// TwinCAT 3 PLC project TF8040_Template_Samples_PLC
// Title: TF8040 Template-Samples
// Company: Beckhoff Automation GmbH
// Author: Beckhoff Automation
// ProjectVersion: 2.0.0.0
// Description: Template-Samples to demonstrate the TF8040 PLC templates.
// ProgramVersion: 3.1.4023.0
// libraries:
//   Tc2_MDP, * (Beckhoff Automation GmbH)
//   Tc2_Standard, * (Beckhoff Automation GmbH)
//   Tc2_SUPS, * (Beckhoff Automation GmbH)
//   Tc2_System, * (Beckhoff Automation GmbH)
//   Tc2_Utilities, * (Beckhoff Automation GmbH)
//   Tc3_BA2, * (Beckhoff Automation GmbH)
//   Tc3_BA2_Common, * (Beckhoff Automation GmbH)
//   Tc3_BACnetRev14, * (Beckhoff Automation GmbH)
//   Tc3_Module, * (Beckhoff Automation GmbH)
//   Tc3_XBA, * (Beckhoff Automation GmbH)
// project tree:
//   / PlcTask.TcTTO (not stored)
//   POUs/ MAIN.TcPOU
//   Templates/DUTs/Enumerations/Building/ E_BA_BuildingMode.TcDUT
//   Templates/DUTs/Enumerations/Plant/AC/ E_BA_AC_OpMod01.TcDUT, E_BA_AC_SelSpErc.TcDUT
//   Templates/DUTs/Enumerations/Universal/ E_BA_EnergyLvl.TcDUT, E_BA_EnergyLvlA.TcDUT, E_BA_MdltCmd.TcDUT, E_BA_OnOff.TcDUT, E_BA_OnOffA.TcDUT
//   Templates/DUTs/Types/Building/ ST_BA_BuildingAlarms.TcDUT
//   Templates/DUTs/Types/General/ ST_BA_GeneralSettings.TcDUT
//   Templates/DUTs/Types/WeatherStation/ ST_BA_WeatherStation.TcDUT
//   Templates/GVLs/ BA2_Param.TcGVL
//   Templates/GVLs/DPAD/Labels/Composition/ LblCmpAC.TcGVL, LblCmpGeneral.TcGVL, LblCmpHeating.TcGVL, LblCmpRoomAutomation.TcGVL, LblUniControl.TcGVL, LblUniFieldDevice.TcGVL
//   Templates/GVLs/EventClasses/ EC_ID.TcGVL
//   Templates/GVLs/Language/English/ LblAggregates_EN.TcGVL, LblControl_EN.TcGVL, LblFunctions_EN.TcGVL, TxtEvent_EN.TcGVL, TxtPlant_EN.TcGVL, TxtTrade_EN.TcGVL
//   Templates/GVLs/Language/German/ LblAggregates_DE.TcGVL, LblControl_DE.TcGVL, LblFunctions_DE.TcGVL, TxtEvent_DE.TcGVL, TxtPlant_DE.TcGVL, TxtTrade_DE.TcGVL
//   Templates/GVLs/Site/ Site.TcGVL
//   Templates/POUs/Trade/AC/Aggregates/Cooler/Temperature/ FB_BA_AC_ColTSuACtrl.TcPOU, FB_BA_AC_ColT_02.TcPOU
//   Templates/POUs/Trade/AC/Aggregates/ERC/ FB_BA_AC_ErcTSuACtrl.TcPOU
//   Templates/POUs/Trade/AC/Aggregates/ERC/Plate/ FB_BA_AC_ErcPl_02.TcPOU
//   Templates/POUs/Trade/AC/Aggregates/PreHeater/ FB_BA_AC_PreHtr.TcPOU, FB_BA_AC_PreHtrTSuACtrl.TcPOU, FB_BA_AC_TRtCtrl.TcPOU
//   Templates/POUs/Trade/AC/ FB_BA_AC.TcPOU
//   Templates/POUs/Trade/AC/General/ FB_BA_AC_OpMod1St.TcPOU, FB_BA_AC_SumNgtCol.TcPOU
//   Templates/POUs/Trade/AC/Plants/ FB_BA_AHU_1st_10.TcPOU
//   Templates/POUs/Trade/AC/Setpoint/Temperature/ FB_BA_AC_SpTRm_01.TcPOU, FB_BA_AC_TCasCtrl_01.TcPOU
//   Templates/POUs/Trade/General/Building/ FB_BA_BuildingAlarms.TcPOU, FB_BA_BuildingGlobal.TcPOU, FB_BA_BuildingMode.TcPOU
//   Templates/POUs/Trade/General/ControlCabinet/ FB_BA_ControlCabinet.TcPOU, FB_BA_ControlCabinetBasic.TcPOU
//   Templates/POUs/Trade/General/EventClasses/ FB_BA_EvtGroups.TcPOU
//   Templates/POUs/Trade/General/ FB_BA_General.TcPOU
//   Templates/POUs/Trade/General/IFP/ FB_BA_IFP.TcPOU
//   Templates/POUs/Trade/General/IFP/Project/ FB_BA_ProjectEx.TcPOU
//   Templates/POUs/Trade/General/Settings/ FB_BA_Settings.TcPOU, FB_BA_WeatherParamter.TcPOU
//   Templates/POUs/Trade/HeatingSystem/Distribution/HeatingCircuit/ FB_BA_H_HtgCir01.TcPOU
//   Templates/POUs/Trade/HeatingSystem/ FB_BA_H.TcPOU
//   Templates/POUs/Trade/HeatingSystem/General/ FB_BA_HtgLmt.TcPOU, FB_BA_H_OpMod.TcPOU
//   Templates/POUs/Trade/HeatingSystem/Setpoint/ FB_BA_H_HtgCir_Sp.TcPOU
//   Templates/POUs/Trade/OutdoorDevices/ FB_BA_OD.TcPOU
//   Templates/POUs/Trade/OutdoorDevices/WeatherStation/ FB_BA_WeatherStation_Draft.TcPOU
//   Templates/POUs/Universal/Aggregat/Analog/ FB_BA_ActuatorAnalog.TcPOU
//   Templates/POUs/Universal/Aggregat/Binary/ FB_BA_ActuatorCmd.TcPOU
//   Templates/POUs/Universal/Control/AntiBlocking/ FB_BA_AntiBlocking.TcPOU
//   Templates/POUs/Universal/Control/EventClasses/ FB_BA_EvtCategory.TcPOU
//   Templates/POUs/Universal/Control/Hysteresis/ FB_BA_Hys_21.TcPOU
//   Templates/POUs/Universal/Control/Monitoring/ FB_BA_FdbAnalog.TcPOU, FB_BA_FdbBinary.TcPOU
//   Templates/POUs/Universal/Control/PID/ FB_BA_PID.TcPOU, FB_BA_PID_Sp.TcPOU
//   Templates/POUs/Universal/Control/Ramp/ FB_BA_RampLimitIncrease.TcPOU
//   Templates/POUs/Universal/Control/Scale/ FB_BA_Scale_02.TcPOU, FB_BA_Scale_04.TcPOU, FB_BA_Scale_04_Y2_3.TcPOU (not stored)
//   Templates/POUs/Universal/Control/TimeDelay/ FB_BA_DlyOff.TcPOU, FB_BA_DlyOn.TcPOU
//   Templates/POUs/Universal/Control/Trend/ FB_BA_TrendLogging.TcPOU
//   Templates/POUs/Universal/Damper/2P/ FB_BA_Dmp2P.TcPOU
//   Templates/POUs/Universal/Motor/1st/ FB_BA_Mot1st.TcPOU
//   Templates/POUs/Universal/Motor/Control/ FB_BA_MotCtlExt.TcPOU
//   Templates/POUs/Universal/Pump/1st/ FB_BA_Pu1st.TcPOU
//   Templates/POUs/Universal/Sensor/ FB_BA_CombinationBI_BV.TcPOU, FB_BA_MeasuredValueCardinal.TcPOU, FB_BA_SensorAnalog.TcPOU, FB_BA_SensorAnalog_IO.TcPOU, FB_BA_SensorBinary.TcPOU, FB_BA_SensorBinary_IO.TcPOU
//   Templates/POUs/Universal/Valve/ FB_BA_Vlv.TcPOU

// ---- Templates/DUTs/Enumerations/Building/E_BA_BuildingMode.TcDUT
{region '#Template'}
	{attribute 'Version' := '1.2.0.0'}
	{attribute 'Tags' := '"LCID": "1031", "Text": "DUT, Building, RA, OpMod, Mode"'}
	{attribute 'Tags' := '"LCID": "1033", "Text": "DUT, Building, RA, OpMod, Mode"'}
	{attribute 'Description' := '"LCID": "1031", "Text": "Gebäude-Betriebsart"'}
	{attribute 'Description' := '"LCID": "1033", "Text": "Building-operation-mode"'}
{endregion}

{attribute qualified_only}
TYPE E_BA_BuildingMode :
(
	eDefault		:= 1,
	eNightWatch		:= 2,
	eCleaning		:= 3
	
) UDINT;
END_TYPE

// ---- Templates/DUTs/Enumerations/Plant/AC/E_BA_AC_OpMod01.TcDUT
{region '#Template'}
	{attribute 'Version' := '1.0.0.0'}
	{attribute 'Tags' := '"LCID": "1031", "Text": "DUT, Plant, AC, OpMod"'}
	{attribute 'Tags' := '"LCID": "1033", "Text": "DUT, Plant, AC, OpMod"'}
	{attribute 'Description' := '"LCID": "1031", "Text": "Betriebsart Klimaanlage"'}
	{attribute 'Description' := '"LCID": "1033", "Text": "Operation Mode Air Conditioning"'}
{endregion}

{attribute qualified_only}
TYPE E_BA_AC_OpMod01 :
(
    Invalid							:= 0,
    eOff							:= 1,	// Aus							// Off
	eOn								:= 2,	// Ein							// On
    eEmergency						:= 3,	// Notfall						// Emergency
    eFrost							:= 4,	// Frost						// Frost
    eSmokeExtractionProgramm		:= 5,	// Entrauchung Programm			// Smoke extraction programm
    eSmokeExtractionSupplyAir		:= 6,	// Entrauchung Zuluft			// Smoke extraction supply air
    eSmokeExtractionExhaustAir		:= 7,	// Entrauchung Fortluft			// Smoke extraction exhaust air
    eFire							:= 8,	// Feuer						// Fire
    eNightCooling					:= 9,	// Nachtkühlung					// Night cooling
    eCoolDownProtection				:= 10,	// Stützbetrieb,Auskühlschutz	// Cool down protection
    eOverHeatingProtection			:= 11,	// Überhitzungsschutz			// Over heating protection
    eAlarm							:= 12,	// Störung						// Alarm
    eForcedVentilation				:= 13,	// Zwangsbelüftung				// Forced ventilation
    eCentralSwitchOff				:= 14	// Zentralabschaltung			// Central switch-off
) UDINT;
END_TYPE

// ---- Templates/DUTs/Enumerations/Plant/AC/E_BA_AC_SelSpErc.TcDUT
{region '#Template'}
	{attribute 'Version' := '1.0.0.0'}
	{attribute 'Tags' := '"LCID": "1031", "Text": "DUT, Plant, AC, Setpoint"'}
	{attribute 'Tags' := '"LCID": "1033", "Text": "DUT, Plant, AC, Setpoint"'}
	{attribute 'Description' := '"LCID": "1031", "Text": "Auswahl Sollwert Energie Rückgewinnung"'}
	{attribute 'Description' := '"LCID": "1033", "Text": "Selection setpoint energy recovery"'}
{endregion}

{attribute 'qualified_only'}
TYPE E_BA_AC_SelSpErc :
(
	eAction				:= 1,	//	E_BA_Action.eDirect = SpCol, E_BA_Action.eReverse = SpHtg, 
	eAverageHtgCol		:= 2	
) UDINT;
END_TYPE

// ---- Templates/DUTs/Enumerations/Universal/E_BA_EnergyLvl.TcDUT
{region '#Template'}
	{attribute 'Version' := '1.0.0.0'}
	{attribute 'Tags' := '"LCID": "1031", "Text": "DUT, Room automation, Heating system"'}
	{attribute 'Tags' := '"LCID": "1033", "Text": "DUT, Room automation, Heating system"'}
	{attribute 'Description' := '"LCID": "1031", "Text": "Betriebsart Energieniveau"'}
	{attribute 'Description' := '"LCID": "1033", "Text": "Operating mode Energy level"'}
{endregion}

{attribute qualified_only}
TYPE E_BA_EnergyLvl :
(
	eProtection		:= 1,
	eEconomy		:= 2,
	eComfort		:= 3
	
) UDINT;
END_TYPE

// ---- Templates/DUTs/Enumerations/Universal/E_BA_EnergyLvlA.TcDUT
{region '#Template'}
	{attribute 'Version' := '1.0.0.0'}
	{attribute 'Tags' := '"LCID": "1031", "Text": "DUT, Room automation, Heating system"'}
	{attribute 'Tags' := '"LCID": "1033", "Text": "DUT, Room automation, Heating system"'}
	{attribute 'Description' := '"LCID": "1031", "Text": "Betriebsart Energieniveau"'}
	{attribute 'Description' := '"LCID": "1033", "Text": "Operating mode Energy level"'}
{endregion}

{attribute qualified_only}
TYPE E_BA_EnergyLvlA :
(
	eAutomatic		:= 1,
	eProtection		:= 2,
	eEconomy		:= 3,
	eComfort		:= 4
	
) UDINT;
END_TYPE

// ---- Templates/DUTs/Enumerations/Universal/E_BA_MdltCmd.TcDUT
{region '#Template'}
	{attribute 'Version' := '1.0.0.0'}
	{attribute 'Tags' := '"LCID": "1031", "Text": "DUT, Operation mode, Universal, Modulation"'}
	{attribute 'Tags' := '"LCID": "1033", "Text": "DUT, Operation mode, Universal, Modulation"'}
	{attribute 'Description' := '"LCID": "1031", "Text": "Modulationsbefehle"'}
	{attribute 'Description' := '"LCID": "1033", "Text": "modulation commands"'}
{endregion}

{attribute 'qualified_only'}
TYPE E_BA_MdltCmd :
(
	eOff			:= 1,
	eOn				:= 2,
	eMin			:= 3,
	eMax			:= 4
	
) UDINT;
END_TYPE

// ---- Templates/DUTs/Enumerations/Universal/E_BA_OnOff.TcDUT
{region '#Template'}
	{attribute 'Version' := '1.0.0.0'}
	{attribute 'Tags' := '"LCID": "1031", "Text": "DUT, Operation mode, Universal, On, Off"'}
	{attribute 'Tags' := '"LCID": "1033", "Text": "DUT, Operation mode, Universal, On, Off"'}
	{attribute 'Description' := '"LCID": "1031", "Text": "Betriebsart Ein Aus"'}
	{attribute 'Description' := '"LCID": "1033", "Text": "Operating on off"'}
{endregion}

{attribute qualified_only}
TYPE E_BA_OnOff :
(
	eOff			:= 1,
	eOn				:= 2
	
) UDINT;
END_TYPE

// ---- Templates/DUTs/Enumerations/Universal/E_BA_OnOffA.TcDUT
{region '#Template'}
	{attribute 'Version' := '1.0.0.0'}
	{attribute 'Tags' := '"LCID": "1031", "Text": "DUT, Operation mode, Universal, On, Off"'}
	{attribute 'Tags' := '"LCID": "1033", "Text": "DUT, Operation mode, Universal, On, Off"'}
	{attribute 'Description' := '"LCID": "1031", "Text": "Betriebsart Ein Aus Auto"'}
	{attribute 'Description' := '"LCID": "1033", "Text": "Operating on off auto"'}
{endregion}

{attribute qualified_only}
TYPE E_BA_OnOffA :
(
	eAutomatic		:= 1,
	eOff			:= 2,
	eOn				:= 3
	
) UDINT;
END_TYPE

// ---- Templates/DUTs/Types/Building/ST_BA_BuildingAlarms.TcDUT
{region '#Template'}
	{attribute 'Version' := '1.2.0.0'}
	{attribute 'Tags' := '"LCID": "1031", "Text": "Types, Publisher, Subscriber, Building, General, Alarms, Events"'}
	{attribute 'Tags' := '"LCID": "1033", "Text": "Types, Publisher, Subscriber, Building, General, Alarms, Events"'}
	{attribute 'Description' := '"LCID": "1031", "Text": "Gebäude-Alarme und -Events"'}
	{attribute 'Description' := '"LCID": "1033", "Text": "Building-alarms and -events"'}
{endregion}
TYPE ST_BA_BuildingAlarms :
STRUCT
	bBurglary				: BOOL;
	bFireAlert				: BOOL;
	bCentralOff				: BOOL;
	bForcedVentilation		: BOOL;
	bSmokeExtraction		: BOOL;
END_STRUCT
END_TYPE

// ---- Templates/DUTs/Types/General/ST_BA_GeneralSettings.TcDUT
{region '#Template'}
	{attribute 'Version' := '1.0.0.0'}
	{attribute 'Tags' := '"LCID": "1031", "Text": "Types, Publisher, Subscriber, AC, General, Settings"'}
	{attribute 'Tags' := '"LCID": "1033", "Text": "Types, Publisher, Subscriber, AC, General, Settings"'}
	{attribute 'Description' := '"LCID": "1031", "Text": "Basis Daten AC"'}
	{attribute 'Description' := '"LCID": "1033", "Text": "Basic data AC"'}
{endregion}
TYPE ST_BA_GeneralSettings :
STRUCT
	fFrostProtectionSetpoint			: REAL;  // frost protection setpoint. for eg. Heating circutis in protection mode
	fTWth								: REAL;  // present value of outside temperature

	fTWthLowLimit						: REAL;  // below this value all frostprotection funcktions in HVAC-Plants will be enabled
	bTWthLowLimit						: BOOL;  // is TRUE when the outside temperature is below the value from fTWthLmtCrit 

	fTWthDamped							: REAL;  // damped outside temperature
	bTWthDampedLowLimit					: BOOL;  // is TRUE when the damped outside temperature is below the value from fTWthLmtCrit 

END_STRUCT
END_TYPE

// ---- Templates/DUTs/Types/WeatherStation/ST_BA_WeatherStation.TcDUT
{region '#Template'}
	{attribute 'Version' := '1.2.0.0'}
	{attribute 'Tags' := '"LCID": "1031", "Text": "Types, Publisher, Subscriber, Weather, Data"'}
	{attribute 'Tags' := '"LCID": "1033", "Text": "Types, Publisher, Subscriber, Weather, Data"'}
	{attribute 'Description' := '"LCID": "1031", "Text": "Daten Wetterstation"'}
	{attribute 'Description' := '"LCID": "1033", "Text": "Weatherstation-data"'}
{endregion}
TYPE ST_BA_WeatherStation :
STRUCT
	bDisturb				: BOOL;
	fLatitude				: REAL;				// [°]
	fLongitude				: REAL;				// [°]
	fSunAzimuth				: REAL;				// [°]
	fSunElevation			: REAL;				// [°]
	bRain					: BOOL;
	stDateTime				: TIMESTRUCT;
	fOutsideTemperature		: REAL;				// [°C]
	fDewPointTemperature	: REAL;				// [°C]		 
	fPressureAbs			: REAL;				// [hPa]
	fPressureRel			: REAL;				// [hPa]			 
	fHumidityAbs			: REAL;				// [g/m³]
	fHumidityRel			: REAL;				// [%rF]	
	fBrightnessNorth		: REAL;				// [Lux]		 
	fBrightnessEast			: REAL;				// [Lux]
	fBrightnessSouth		: REAL;				// [Lux]
	fBrightnessWest			: REAL;				// [Lux]			 
	fDawn					: REAL;				// [Lux] 
	fGlobalRadiation		: REAL;				// [W/m²]			 
	fWindDirection			: REAL;				// [°]
	fWindSpeed				: REAL;				// [m/s]
END_STRUCT
END_TYPE

// ---- Templates/GVLs/BA2_Param.TcGVL
{region '#Template'}
	{attribute 'Version' := '0.0.1.0'}
	{attribute 'Tags' := '"LCID": "1031", "Text": "GVL, Constants"'}
	{attribute 'Tags' := '"LCID": "1033", "Text": "GVL, Constants"'}
	{attribute 'Description' := '"LCID": "1031", "Text": "Globale Konstanten"'}
	{attribute 'Description' := '"LCID": "1033", "Text": "Global constants"'}
{endregion}

{attribute 'qualified_only'}
{attribute 'strict'}
VAR_GLOBAL CONSTANT 
	fAP                					: REAL 						:= 1013.25;	// Hydrostatischer Luftdruck	//	atmospheric pressure

	nDefTimeDelay_ToAbnormal			: UDINT						:= 1;
	nDefTimeDelay_ToNormal				: UDINT						:= 0;

	fDefCOVIncrement					: REAL						:= 0.1;	

	fDefLimitDeadband					: REAL						:= 0.0;

	nLoop_DefOpMode						: E_BA_PIDMode				:= E_BA_PIDMode.eP1ID;	
	
	{warning disable C0228}
	stTrend_DefStartTime				: ST_BA_DateTime			;(*:= F_BA_ToSTDateTime(DT#2099-01-01-00:13);*)
	stTrend_DefStopTime					: ST_BA_DateTime			;(* := F_BA_ToSTDateTime(DT#2099-01-01-00:13);*)
	{warning restore C0228}
	nTrend_BufferSize					: UDINT						:= 500;	// Count of entries in a Trend-Buffer	
	bTrend_DefLogEnable					: BOOL						:= FALSE;
	bTrend_DefStopOnFull				: BOOL						:= FALSE;
	nTrend_DefLogInterval				: UDINT						:= 90;	// (in [s])
	nTrend_DefNotificationThreshold		: UDINT						:= 50;
	eTrend_DefLoggingType				: E_BA_LoggingType			:= E_BA_LoggingType.ePolled;				
END_VAR

// ---- Templates/GVLs/DPAD/Labels/Composition/LblCmpAC.TcGVL
{region '#Template'}
	{attribute 'Version' := '1.2.0.0'}
	{attribute 'Tags' := '"LCID": "1031", "Text": "GVL, AC, AKS, Plants, ObjectName, Description"'}
	{attribute 'Tags' := '"LCID": "1033", "Text": "GVL, AC, DPAD, Plants, ObjectName, Description"'}
	{attribute 'Description' := '"LCID": "1031", "Text": "Anlagenkennzeichnungssystem, AC Labels Kompensation"'}
	{attribute 'Description' := '"LCID": "1033", "Text": "Data Point Addressing Description, AC labels compensation"'}
{endregion}

{attribute 'qualified_only'}
VAR_GLOBAL
///////////////////////
//	Aggregates\Cooler	
	Cooler_TFl							:FB_BA_Label	:= LblAggregates_TemperatureFlow;	
	Cooler_TRt							:FB_BA_Label	:= LblAggregates_TemperatureReturnFlow;	

	Cooler_TSuACtrl						:FB_BA_Label	:= LblControl_SupplyAirTemperatureControl;
	Cooler_TSuACtrl_Ctrl				:FB_BA_Label	:= LblFunctions_LoopObject; 
	Cooler_TSuALimitationCtrl			:FB_BA_Label	:= LblControl_SupplyAirTemperatureLimitationControl;

	Cooler_XSuACtrl						:FB_BA_Label	:= LblControl_SupplyAirDehumidifierControl; 
	Cooler_XSuACtrl_Ctrl				:FB_BA_Label	:= LblFunctions_LoopObject; 
	Cooler_Dehumf						:FB_BA_Label	:= LblControl_OperationalMessageDehumidification;	

	Cooler_Vlv							:FB_BA_Label	:= LblAggregates_Valve;
	Cooler_Pu							:FB_BA_Label	:= LblAggregates_Pump;
	
//	Aggregates\ERC
	ERC_DiffPrssSwi						:FB_BA_Label	:= LblAggregates_PressureDifferential;												 										 
	ERC_IcePrtcRamp						:FB_BA_Label	:= LblControl_EnergyRecoveryDeicingRamp;
	ERC_Motor							:FB_BA_Label	:= LblAggregates_HeatRecovery;
	ERC_TExhACtrl						:FB_BA_Label	:= LblControl_ExhaustAirTemperatureControl;
	ERC_TSuACtrl						:FB_BA_Label	:= LblControl_SupplyAirTemperatureControl;
	ERC_TSuACtrl_Ctrl					:FB_BA_Label	:= LblFunctions_LoopObject; 

	ERC_DiffPrssSensor					:FB_BA_Label	:= LblAggregates_PressureDifferential;	
	ERC_Damping							:FB_BA_Label	:= LblAggregates_PressureDifferential;
	ERC_IcePrtcDiffPrssCtrl				:FB_BA_Label	:= LblControl_ExhaustAirTemperatureControl;
	ERC_Dmp								:FB_BA_Label	:= LblAggregates_VentilationDamperSupplyAir;	
	ERC_ByDmp							:FB_BA_Label	:= LblAggregates_VentilationDamperBypassAir;

//	Aggregates\Humidifier
	Humf_HuDet							:FB_BA_Label	:= LblAggregates_Hygrostat;	
	Humf_XSuACtrl						:FB_BA_Label	:= LblControl_SupplyAirHumidifierController;
	Humf_XSuACtrl_Ctrl					:FB_BA_Label	:= LblFunctions_LoopObject;
	Humf_Motor							:FB_BA_Label	:= LblAggregates_Humidifier;
	Humf_DlyOff							:FB_BA_Label	:= LblControl_DelayOff;	
	Humf_HLmtCtrl						:FB_BA_Label	:= LblControl_HumidityLimitationControl;

//	Aggregates\MixedAir
	Mix_TSuACtrl						:FB_BA_Label	:= LblControl_SupplyAirTemperatureControl;
	Mix_TSuACtrl_Ctrl					:FB_BA_Label	:= LblFunctions_LoopObject; 
	Mix_StartUpRamp						:FB_BA_Label	:= LblControl_MixedAirStartUpRamp;
	Mix_DmpMixA							:FB_BA_Label	:= LblAggregates_VentilationDamperMixAir;	
	Mix_DmpOuA							:FB_BA_Label	:= LblAggregates_VentilationDamperOutsideAir;	
	Mix_DmpExhA							:FB_BA_Label	:= LblAggregates_VentilationDamperExhaustAir;	

//	Aggregates\pre-heater
	PreHtr_TFl							:FB_BA_Label	:= LblAggregates_TemperatureFlow;	
	PreHtr_TRt							:FB_BA_Label	:= LblAggregates_TemperatureReturnFlow;	
	PreHtr_TSuACtrl						:FB_BA_Label	:= LblControl_SupplyAirTemperatureControl;
	PreHtr_TSuACtrl_Ctrl				:FB_BA_Label	:= LblFunctions_LoopObject; 
	PreHtr_TFrost						:FB_BA_Label	:= LblControl_TemperatureFrost;	
	PreHtr_TFrostPrtcCtrlAir			:FB_BA_Label	:= LblControl_FrostProtectionControl;
	PreHtr_FrostThermostat				:FB_BA_Label	:= LblAggregates_FrostProtectionMonitor;												 										 
	PreHtr_FrostThermostat_Input		:FB_BA_Label	:= LblFunctions_DangerAlarm;
	PreHtr_Vlv							:FB_BA_Label	:= LblAggregates_Valve;
	PreHtr_Pu							:FB_BA_Label	:= LblAggregates_Pump;		
	PreHtr_TRtCtrl						:FB_BA_Label	:= LblControl_ReturnWaterControl;
	PreHtr_TRtCtrl_SpTRtW				:FB_BA_Label	:= LblFunctions_Setpoint;
	PreHtr_TRtCtrl_PreRinseDelay		:FB_BA_Label	:= LblControl_DelayOn;
	PreHtr_TRtCtrl_PreRinseDelay_TiDly	:FB_BA_Label	:= LblControl_PreRinseDuration;
	PreHtr_TRtCtrl_PreRinseDst			:FB_BA_Label	:= LblControl_DisturbancePreRinse;	 								 
	PreHtr_TRtCtrl_PreRinseSp			:FB_BA_Label	:= LblControl_CalculationPreRinseSetpoint;			
	PreHtr_TRtCtrl_Ctrl					:FB_BA_Label	:= LblFunctions_LoopObject; 		
	
	PreHtr_ProcessPreRinse				:FB_BA_LabelProcess	:= LblControl_ProcPreRinse;

//	Aggregates\re-heater
	ReHtr_TFl							:FB_BA_Label	:= LblAggregates_TemperatureFlow;	
	ReHtr_TRt							:FB_BA_Label	:= LblAggregates_TemperatureReturnFlow;	
	ReHtr_TSuACtrl						:FB_BA_Label	:= LblControl_SupplyAirTemperatureControl;
	ReHtr_TSuACtrl_Ctrl					:FB_BA_Label	:= LblFunctions_LoopObject;
	ReHtr_TMinSuACtrl					:FB_BA_Label	:= LblControl_SupplyAirTemperatureLimitationControl;
 
	ReHtr_Vlv							:FB_BA_Label	:= LblAggregates_Valve;
	ReHtr_Pu							:FB_BA_Label	:= LblAggregates_Pump;		
		
///////////////////////
//	General
	General_OpModMan					:FB_BA_Label	:= LblControl_OperationModeSelection;							
	General_Sched						:FB_BA_Label	:= LblFunctions_Scheduler;							
	General_OpModPr						:FB_BA_Label	:= LblControl_PresentOperationMode;		
	
//	Summer night cooling
	General_SumNgtCol_WthTLoLmt			:FB_BA_Label	:= LblControl_OutsideTemperatureLowLimit;			
	General_SumNgtCol_RmTHys			:FB_BA_Label	:= LblControl_HysteresisRoomTemperature;			
	General_SumNgtCol_SwiOnDiffT		:FB_BA_Label	:= LblControl_OnValueDifferenceOutsideInsightTemperature;			
	General_SumNgtCol_SwiOffDiffT		:FB_BA_Label	:= LblControl_OffValueDifferenceOutsideInsightTemperature;			
	General_SumNgtCol_Q					:FB_BA_Label	:= LblFunctions_OperationalMessage;												 
	General_SumNgtCol_Sched				:FB_BA_Label	:= LblFunctions_Scheduler;		
///////////////////////
//	Setpoint\Temperature
	SpTRm_X1							:FB_BA_Label	:= LblControl_X01;	
	SpTRm_X2							:FB_BA_Label	:= LblControl_X02;	
	SpTRm_X3							:FB_BA_Label	:= LblControl_X03;	
	SpTRm_X4							:FB_BA_Label	:= LblControl_X04;	
	
	SpTRm_Y1							:FB_BA_Label	:= LblControl_Y01;
	SpTRm_Y2_3							:FB_BA_Label	:= LblControl_Y02_03;
	SpTRm_Y4							:FB_BA_Label	:= LblControl_Y03;
	SpTRm_Sp							:FB_BA_Label	:= LblFunctions_SetpointCalculated;
	
	SpTRm_SpColX1						:FB_BA_Label	:= LblControl_SummerCompensationX1;	
	SpTRm_SpColX2						:FB_BA_Label	:= LblControl_SummerCompensationX2;	
	SpTRm_SpColY1						:FB_BA_Label	:= LblControl_SummerCompensationY1;	
	SpTRm_SpColY2						:FB_BA_Label	:= LblControl_SummerCompensationY2;	
	SpTRm_SpColYMin						:FB_BA_Label	:= LblControl_SummerCompensationYmin;
	SpTRm_SpColYMax						:FB_BA_Label	:= LblControl_SummerCompensationYmax;	
	SpTRm_SpCol							:FB_BA_Label	:= LblControl_SummerCompensationSp;	
	
	SpTRm_SpHtgX1						:FB_BA_Label	:= LblControl_WinterCompensationX1;	
	SpTRm_SpHtgX2						:FB_BA_Label	:= LblControl_WinterCompensationX2;	
	SpTRm_SpHtgY1						:FB_BA_Label	:= LblControl_WinterCompensationY1;	
	SpTRm_SpHtgY2						:FB_BA_Label	:= LblControl_WinterCompensationY2;	
	SpTRm_SpHtgYMin						:FB_BA_Label	:= LblControl_WinterCompensationYmin;
	SpTRm_SpHtgYMax						:FB_BA_Label	:= LblControl_WinterCompensationYmax;		
	SpTRm_SpHtg							:FB_BA_Label	:= LblControl_WinterCompensationSp;	
	
	SpTSuA_SelSpErc						:FB_BA_Label	:= LblControl_OperationModeSelection;							
	SpTSuA_SpErc						:FB_BA_Label	:= LblFunctions_SetpointCalculated;	

	TCasCtrl_SpHtg						:FB_BA_Label	:= LblControl_SuppyAirTempSetpointHeaterCalc;			
	TCasCtrl_SpCol						:FB_BA_Label	:= LblControl_SuppyAirTempSetpointCoolerCalc;			
	TCasCtrl_SpErc						:FB_BA_Label	:= LblControl_SuppyAirTempSetpointERCCalc;			
	TCasCtrl_Ctrl						:FB_BA_Label	:= LblFunctions_LoopObjectCascadeSupplyAirTemperature; 			
	TCasCtrl_SelSpErc					:FB_BA_Label	:= LblControl_OperationModeSelection;							
//	Setpoint\Humidity
	HumCasCtrl_Ctrl						:FB_BA_Label	:= LblFunctions_LoopObjectCascadeSupplyAirHumidity; 	
	SpHum_SpH							:FB_BA_Label	:= LblControl_SetpointRelHumidity;			
	SpHum_SpX							:FB_BA_Label	:= LblControl_SetpointAbsHumidity;
	SpHum_SpHHumf						:FB_BA_Label	:= LblControl_SetpointRelHumidityHumidification;			
	SpHum_SpHDehumf						:FB_BA_Label	:= LblControl_SetpointRelHumidityDehumidification;			
	SpHum_SpXHumf						:FB_BA_Label	:= LblControl_SetpointAbsHumidityHumidification;	
	SpHum_SpXDehumf						:FB_BA_Label	:= LblControl_SetpointAbsHumidityDehumidification;
//	
	PlantControlStatus   	:FB_BA_Label2x :=(iAggregate:=LblControl_PlantControl,		iFunction:=LblFunctions_Status);
	TSequenceControlStatus  :FB_BA_Label2x :=(iAggregate:=LblControl_TSequenceControl,	iFunction:=LblFunctions_Status);		
	HSequenceControlStatus  :FB_BA_Label2x :=(iAggregate:=LblControl_HSequenceControl,	iFunction:=LblFunctions_Status);		
//	AHU	
	AHU_TOuA						:FB_BA_Label	:= LblAggregates_TemperatureOutside;
	AHU_HOuA						:FB_BA_Label	:= LblAggregates_RelativeHumidityOutsideAir;
	AHU_XOuA						:FB_BA_Label	:= LblAggregates_AbsoluteHumidtiyOutsideAir;
	AHU_TExhA						:FB_BA_Label	:= LblAggregates_TemperatureExhaustAir;	
	AHU_HExhA						:FB_BA_Label	:= LblAggregates_RelativeHumidityExhaustAir;	
	AHU_XExhA						:FB_BA_Label	:= LblAggregates_AbsoluteHumidtiyExhaustAir;	
	AHU_TSuA						:FB_BA_Label	:= LblAggregates_TemperatureSupplyAir;	
	AHU_HSuA						:FB_BA_Label	:= LblAggregates_RelativeHumiditySupplyAir;	
	AHU_XSuA						:FB_BA_Label	:= LblAggregates_AbsoluteHumiditySupplyAir;	
	AHU_TExtA						:FB_BA_Label	:= LblAggregates_TemperatureExtractAir;	
	AHU_HExtA						:FB_BA_Label	:= LblAggregates_RelativeHumiditiyExtractAir;	
	AHU_XExtA						:FB_BA_Label	:= LblAggregates_AbsoluteHumidityExtractAir;	
	AHU_TRm							:FB_BA_Label	:= LblAggregates_TemperatureRoomAir;	
	AHU_HRm							:FB_BA_Label	:= LblAggregates_RelativeHumidityRoomHumidity;	
	AHU_XRm							:FB_BA_Label	:= LblAggregates_AbsoluteHumidityRoomAir;	
	AHU_DiffPrssOuAFilt				:FB_BA_Label	:= LblAggregates_PressureDifferentialOutsideAirFilter;	
	AHU_FiltOuAMonit				:FB_BA_Label	:= LblAggregates_AirFilterOutsideAir;
	AHU_DiffPrssExtAFilt			:FB_BA_Label	:= LblAggregates_PressureDifferentialExtractAirFilter;	
	AHU_FiltExtAMonit				:FB_BA_Label	:= LblAggregates_AirFilterExtractAir;
	AHU_SumNgtCol					:FB_BA_Label	:= LblControl_SummerNightCooling;
	AHU_OpMod						:FB_BA_Label	:= LblControl_OperationMode;
	AHU_OuADmp						:FB_BA_Label	:= LblAggregates_VentilationDamperOutsideAir;
	AHU_SuAPrss						:FB_BA_Label	:= LblAggregates_PressureSupplyAir;	
	AHU_SuADiffPrss					:FB_BA_Label	:= LblAggregates_PressureDifferentialSupplyAirFan;	
	AHU_SuAFan						:FB_BA_Label	:= LblAggregates_FanSupplyAir;
	AHU_SuADiffPrssMonit			:FB_BA_Label	:= LblControl_DifferencePressureMonitoringSupplyAirFan;
	AHU_ExhADmp						:FB_BA_Label	:= LblAggregates_VentilationDamperExhaustAir;
	AHU_ExtAPrss					:FB_BA_Label	:= LblAggregates_PressureExtractAir;	
	AHU_ExtADiffPrss				:FB_BA_Label	:= LblAggregates_PressureDifferentialExtractAirFan;	
	AHU_ExtAFan						:FB_BA_Label	:= LblAggregates_FanExtractAir;
	AHU_ExtADiffPrssMonit			:FB_BA_Label	:= LblControl_DifferencePressureMonitoringExtractAirFan;
	AHU_SpTRm						:FB_BA_Label	:= LblControl_TSetpointCalculation;
	AHU_TCasCtrl					:FB_BA_Label	:= LblControl_TCascadeSupplyAirControl;
	AHU_TSeqLink					:FB_BA_Label2x	:= TSequenceControlStatus;
	AHU_SpHRm						:FB_BA_Label	:= LblControl_HSetpointCalculation;
	AHU_HCasCtrl					:FB_BA_Label	:= LblControl_HCascadeSupplyAirControl;
	AHU_HSeqLink					:FB_BA_Label2x	:= HSequenceControlStatus;	
	AHU_ReHtr						:FB_BA_Label	:= LblControl_ReHeater;
	AHU_PreHtr						:FB_BA_Label	:= LblControl_PreHeater;
	AHU_Erc							:FB_BA_Label	:= LblControl_EnergyRecovery;
	AHU_Col							:FB_BA_Label	:= LblControl_Cooler;
	AHU_Humf						:FB_BA_Label	:= LblAggregates_Humidifier;
	AHU_PlantCtrl					:FB_BA_Label2x	:= PlantControlStatus;	
END_VAR

// ---- Templates/GVLs/DPAD/Labels/Composition/LblCmpGeneral.TcGVL
{region '#Template'}
	{attribute 'Version' := '1.2.0.0'}
	{attribute 'Tags' := '"LCID": "1031", "Text": "GVL, General, AKS, Plants, ObjectName, Description"'}
	{attribute 'Tags' := '"LCID": "1033", "Text": "GVL, General, DPAD, Plants, ObjectName, Description"'}
	{attribute 'Description' := '"LCID": "1031", "Text": "Anlagenkennzeichnungssystem, Allgemein Labels Kompensation"'}
	{attribute 'Description' := '"LCID": "1033", "Text": "Data Point Addressing Description, General labels compensation"'}
{endregion}

{attribute 'qualified_only'}
VAR_GLOBAL
	BuildingAlarms_FireAlert						: FB_BA_Label := LblControl_FireAlert;
	BuildingAlarms_Bgly								: FB_BA_Label := LblControl_Burglary;
	BuildingAlarms_CentSwiOff						: FB_BA_Label := LblControl_CentralSwitchOff;
                                  				
	BuildingMode_OpModMan							: FB_BA_Label := LblControl_BuildingModeManual;
	BuildingMode_OpModPr							: FB_BA_Label := LblControl_BuildingModeActual;
	BuildingMode_Sched								: FB_BA_Label := LblControl_BuildingModeSched;
                                  				
	BuildingGlobal_BuildAlm							: FB_BA_Label := LblControl_BuildingAlarms;
	BuildingGlobal_BuildMode						: FB_BA_Label := LblControl_BuildingMode;
	
	ControlCabinet_Fuse								: FB_BA_Label := LblControl_Fuse;	
	ControlCabinet_Fuse_Input						: FB_BA_Label := LblFunctions_Fault;	
	ControlCabinet_LampFault						: FB_BA_Label := LblControl_EventIndicationLamp;			
	ControlCabinet_LampFault_Cmd					: FB_BA_Label := LblFunctions_SwitchingCommand;			
	ControlCabinet_AckButton 						: FB_BA_Label := LblControl_Acknowledge;	
	ControlCabinet_AckButton_Input					: FB_BA_Label := LblControl_ButtonLocalAcknowledgement;
	ControlCabinet_AckButton_Value					: FB_BA_Label := LblControl_ButtonRemoteAcknowledgement;
	ControlCabinet_RstHw							: FB_BA_Label := LblControl_AcknowledgeCommand;			
	ControlCabinet_RstHw_Cmd						: FB_BA_Label := LblFunctions_SwitchingCommand;	

	EvtGroups_LifeSafety							: FB_BA_Label := LblControl_EvtCategoryLifeSafty;									  
	EvtGroups_SaftyMessage							: FB_BA_Label := LblControl_EvtCategorySaftyMessage;									  
	EvtGroups_AlarmMessage							: FB_BA_Label := LblControl_EvtCategoryAlarmMessage;									  
	EvtGroups_FaultMessage							: FB_BA_Label := LblControl_EvtCategoryFaultMessage;									  
	EvtGroups_MaintenanceMessage					: FB_BA_Label := LblControl_EvtCategoryMaintenanceMessage;									  
	EvtGroups_System								: FB_BA_Label := LblControl_EvtCategorySystem;									  
	EvtGroups_ManualOperation						: FB_BA_Label := LblControl_EvtCategoryManualOperation;									  
	EvtGroups_Other									: FB_BA_Label := LblControl_EvtCategoryOther;									  
	
	Settings_WthParam								: FB_BA_Label := LblControl_WeatherParameters;	
	
	WthParam_SpFrstProtec							: FB_BA_Label := LblControl_SetpointFrostProtection;
	WthParam_TWthLowLimitVal						: FB_BA_Label := LblControl_SetpointMinimumOutsideTemperature;
	WthParam_TWthLowLimit							: FB_BA_Label := LblControl_OperationalMessageTemperatureWeatherLowLimit;	
	WthParam_TWthDamped								: FB_BA_Label := LblControl_MeanDamped;
	WthParam_TWthDampedLowLimit						: FB_BA_Label := LblControl_OperationalMessageTemperatureWeatherDampedLowLimit;	
END_VAR

// ---- Templates/GVLs/DPAD/Labels/Composition/LblCmpHeating.TcGVL
{region '#Template'}
	{attribute 'Version' := '1.2.0.0'}
	{attribute 'Tags' := '"LCID": "1031", "Text": "GVL, Heating, AKS, Plants, ObjectName, Description"'}
	{attribute 'Tags' := '"LCID": "1033", "Text": "GVL, Heating, DPAD, Plants, ObjectName, Description"'}
	{attribute 'Description' := '"LCID": "1031", "Text": "Anlagenkennzeichnungssystem, Heizsystem Labels Kompensation"'}
	{attribute 'Description' := '"LCID": "1033", "Text": "Data Point Addressing Description, Heating system labels compensation"'}
{endregion}

{attribute 'qualified_only'}
VAR_GLOBAL
	H_HtgCir_Sp_NgtOffs						:FB_BA_Label	:= LblControl_OffsetNightSetpoint;
	H_HtgCir_Sp_SpFlWT						:FB_BA_Label	:= LblFunctions_Setpoint;
	H_HtgCir_Sp_HtgCrv						:FB_BA_Label	:= LblControl_HeatingCurve;
	H_OpMod_OpModMan						:FB_BA_Label	:= LblControl_OperationModeSelection;
	H_OpMod_Sched							:FB_BA_Label	:= LblFunctions_Scheduler;
	H_OpMod_OpModPr							:FB_BA_Label	:= LblControl_PresentOperationMode;
	H_OpMod_Rls								:FB_BA_Label	:= LblFunctions_Enabled;
	
	HtgLmt_Sp								:FB_BA_Label	:= LblFunctions_Setpoint;
	HtgLmt_Q								:FB_BA_Label	:= LblFunctions_OperationalMessage;
	
	
	H_HtgCir_TFl						:FB_BA_Label	:= LblAggregates_TemperatureFlow;
	H_HtgCir_TRt						:FB_BA_Label	:= LblAggregates_TemperatureReturnFlow;
	H_HtgCir_Vlv						:FB_BA_Label	:= LblAggregates_Valve;
	H_HtgCir_Pu							:FB_BA_Label	:= LblAggregates_Pump;
	H_HtgCir_Sp							:FB_BA_Label	:= LblControl_SetpointGeneration;
	H_HtgCir_OpMod						:FB_BA_Label	:= LblControl_OperationMode;
	H_HtgCir_TFlCtrl					:FB_BA_Label	:= LblControl_FlowTemperatureControl;
	H_HtgCir_HtgLmt						:FB_BA_Label	:= LblControl_HeatingLimit;			
END_VAR

// ---- Templates/GVLs/DPAD/Labels/Composition/LblCmpRoomAutomation.TcGVL
{region '#Template'}
	{attribute 'Version' := '1.2.0.0'}
	{attribute 'Tags' := '"LCID": "1031", "Text": "GVL, Room automation, AKS, Plants, ObjectName, Description"'}
	{attribute 'Tags' := '"LCID": "1033", "Text": "GVL, Room automation, DPAD, Plants, ObjectName, Description"'}
	{attribute 'Description' := '"LCID": "1031", "Text": "Anlagenkennzeichnungssystem, Raum Automation Labels Kompensation"'}
	{attribute 'Description' := '"LCID": "1033", "Text": "Data Point Addressing Description, Room automation labels compensation"'}
{endregion}

{attribute 'qualified_only'}
VAR_GLOBAL
	BuildingEnergyLevel_EnergLvlMan					: FB_BA_Label := LblControl_BuildingEnergyLevelManual;
	BuildingEnergyLevel_EnergLvlPr					: FB_BA_Label := LblControl_BuildingEnergyLevelActual;
	BuildingEnergyLevel_Sched						: FB_BA_Label := LblControl_BuildingEnergyLevelSched;
    
	BuildingSpRmT_SumCpsn							: FB_BA_Label := LblControl_SummerCompensation;
	BuildingSpRmT_WinCpsn							: FB_BA_Label := LblControl_WinterCompensation;
	BuildingSpRmT_PrtcHtg							: FB_BA_Label := LblFunctions_SetpointProtectionHeating;
	BuildingSpRmT_EcoHtg							: FB_BA_Label := LblFunctions_SetpointEconomyHeating;
	BuildingSpRmT_PreCmfHtg							: FB_BA_Label := LblFunctions_SetpointPreComfortHeating;
	BuildingSpRmT_CmfHtg							: FB_BA_Label := LblFunctions_SetpointComfortHeating;
	BuildingSpRmT_PrtcCol							: FB_BA_Label := LblFunctions_SetpointProtectionCooling;
	BuildingSpRmT_EcoCol							: FB_BA_Label := LblFunctions_SetpointEconomyCooling;
	BuildingSpRmT_PreCmfCol							: FB_BA_Label := LblFunctions_SetpointPreComfortCooling;
	BuildingSpRmT_CmfCol							: FB_BA_Label := LblFunctions_SetpointComfortCooling;
	BuildingSpRmT_ShiftHtg							: FB_BA_Label := LblControl_SetpointShiftHeating;
	BuildingSpRmT_ShiftCol							: FB_BA_Label := LblControl_SetpointShiftCooling;
	
	BuildingSunprotection_SpIce						: FB_BA_Label := LblControl_SetpointIce;
	BuildingSunprotection_SunPrtcPosIntval			: FB_BA_Label := LblControl_SunProtectionInterval;
	BuildingSunprotection_DeiceTi					: FB_BA_Label := LblControl_DeiceTime;
	BuildingSunprotection_GlobalThAutoValOn			: FB_BA_Label := LblControl_GlobalThermoAutomaticValueOn;
	BuildingSunprotection_GlobalThAutoValOff		: FB_BA_Label := LblControl_GlobalThermoAutomaticValueOff;
	BuildingSunprotection_GlobalTwiLgtAutoValOn		: FB_BA_Label := LblControl_GlobalTwilightAutomaticValueOn;
	BuildingSunprotection_GlobalTwiLgtAutoValOff	: FB_BA_Label := LblControl_GlobalTwilightAutomaticValueOff;
	BuildingSunprotection_IceAlert					: FB_BA_Label := LblControl_IceAlert;
	BuildingSunprotection_GlobalThAutoRlse			: FB_BA_Label := LblControl_GlobalThermoAutomaticRelease;
	BuildingSunprotection_GlobalTwiLgtAutoRlse		: FB_BA_Label := LblControl_GlobalTwilightAutomaticRelease;
	BuildingSunprotection_GlobalResetManMode		: FB_BA_Label := LblControl_GlobalResetManMode;
	
	Facade_DlyStrmOn								: FB_BA_Label := LblControl_TimeDelayStormOn;
	Facade_DlyStrmOff								: FB_BA_Label := LblControl_TimeDelayStormOff;
	Facade_MntnEn									: FB_BA_Label := LblControl_MaintenanceEnable;                    		
	Facade_MntnPos									: FB_BA_Label := LblControl_MaintenancePosition;
	Facade_MntnAngl									: FB_BA_Label := LblControl_MaintenanceAngle;
	Facade_FcdThAutoEn								: FB_BA_Label := LblControl_FacadeThermoAutomaticEnable;
	Facade_FcdThAutoColPos							: FB_BA_Label := LblControl_FacadeThermoAutomaticCoolingPosition;
	Facade_FcdThAutoColAngl							: FB_BA_Label := LblControl_FacadeThermoAutomaticCoolingAngle;
	Facade_FcdTwiLgtAutoEn							: FB_BA_Label := LblControl_FacadeTwilightAutomaticEnable;
	Facade_SunPrtcValOn								: FB_BA_Label := LblControl_SunProtectionValueOn;
	Facade_SunPrtcValOff							: FB_BA_Label := LblControl_SunProtectionValueOff;
	Facade_SunPrtcDlyOn								: FB_BA_Label := LblControl_TimeDelaySunProtectionOn;
	Facade_SunPrtcDlyOff							: FB_BA_Label := LblControl_TimeDelaySunProtectionOff;
	Facade_FcdParkEn								: FB_BA_Label := LblControl_FacadeParkingEnable;
	Facade_FcdParkPos								: FB_BA_Label := LblControl_FacadeParkingPosition;
	Facade_FcdParkAngl								: FB_BA_Label := LblControl_FacadeParkingAngle;
	Facade_WndPrtcState								: FB_BA_Label := LblControl_WindProtectionState;
	Facade_SunPrtcState								: FB_BA_Label := LblControl_SunProtectionState;
    
	SunBld_LocInputPos								: FB_BA_Label := LblControl_SetpointSunblindPosition;
	SunBld_LocInputAngl								: FB_BA_Label := LblControl_SetpointSunblindAngle;
	SunBld_LocButtonStart							: FB_BA_Label := LblControl_CommandSunblindStart;
	SunBld_ActlPos									: FB_BA_Label := LblControl_FeedbackSunblindPosition;
	SunBld_ActlAngl									: FB_BA_Label := LblControl_FeedbackSunblindAngle;
	SunBld_ActlPrio									: FB_BA_Label := LblControl_FeedbackSunblindPrio;
	SunBld_ManSwi									: FB_BA_Label := LblControl_ButtonSunblind;
		
	HeatCoolAxisAnlg_RmTSen							: FB_BA_Label := LblAggregates_TemperatureRoomAir;
	HeatCoolAxisAnlg_RmTAdj							: FB_BA_Label := LblAggregates_RoomControlUnit;
	HeatCoolAxisAnlg_PrtcDetc						: FB_BA_Label := LblAggregates_PresenceSwitches;
	HeatCoolAxisAnlg_WdwCon							: FB_BA_Label := LblAggregates_WindowContact;
	HeatCoolAxisAnlg_VlvHtg							: FB_BA_Label :=(sObjName:='VEN',sDescr:='Heizventil');
 	HeatCoolAxisAnlg_VlvCol							: FB_BA_Label :=(sObjName:='VEN',sDescr:='Kuehlventil');
 	HeatCoolAxisAnlg_Ctrl							: FB_BA_Label := LblControl_RoomTemperatureControl;
 	HeatCoolAxisAnlg_Ctrl_CtrlHtg					: FB_BA_Label :=(sObjName:='LPH',sDescr:='Heizregler');
 	HeatCoolAxisAnlg_Ctrl_CtrlCol					: FB_BA_Label :=(sObjName:='LPC',sDescr:='Kuehlregler');
	HeatCoolAxisAnlg_DewPoint						: FB_BA_Label := LblAggregates_MonitorDewPoint;

	SunBldZone_SunBld								: FB_BA_Label := LblAggregates_Blind;
                                          	
//	RoomAutomation_RoomGeneral						: FB_BA_Label := LabelPlants.Room_automation;
	
	RoomGeneral_FcdEast								: FB_BA_Label := LblControl_Facade;
END_VAR

// ---- Templates/GVLs/DPAD/Labels/Composition/LblUniControl.TcGVL
{region '#Template'}
	{attribute 'Version' := '1.2.0.0'}
	{attribute 'Tags' := '"LCID": "1031", "Text": "GVL, Universal, AKS, Plants, ObjectName, Description"'}
	{attribute 'Tags' := '"LCID": "1033", "Text": "GVL, Universal, DPAD, Plants, ObjectName, Description"'}
	{attribute 'Description' := '"LCID": "1031", "Text": "Anlagenkennzeichnungssystem, Universal Labels Kompensation"'}
	{attribute 'Description' := '"LCID": "1033", "Text": "Data Point Addressing Description, Universal labels compensation"'}
{endregion}

{attribute 'qualified_only'}
VAR_GLOBAL
//	Anti blocking
	Analog3Pnt_HysPos					:FB_BA_Label	:= LblFunctions_Hysteresis;
	Analog3Pnt_TimeOpen     			:FB_BA_Label	:= LblControl_DriveTimeOpen;	
	Analog3Pnt_TimeCls					:FB_BA_Label	:= LblControl_DriveTimeClose;
	Analog3Pnt_Pos						:FB_BA_Label	:= LblFunctions_ControlSignal;	
//	Anti blocking
	AntiBlocking_IdlePeriod				:FB_BA_Label	:= LblControl_IdlePeriod;
	AntiBlocking_ImpulsLength           :FB_BA_Label	:= LblControl_ImpulsLength;	
//	Continuous steps	
	ContinuousSteps_SwitchOn				:FB_BA_Label	:= LblFunctions_Threshold;
	ContinuousSteps_Hysteresis			:FB_BA_Label	:= LblFunctions_Hysteresis;
//	Delay
	DelayOn_TiDly						:FB_BA_Label	:= LblControl_TimeDelay;
	DelayOff_TiDly						:FB_BA_Label	:= LblControl_TimeDelay;
//	Hysteresis	
	Hysteresis_On						:FB_BA_Label	:= LblFunctions_LimitMAX;
	Hysteresis_Off						:FB_BA_Label	:= LblFunctions_LimitMIN;
	Hysteresis_Q						:FB_BA_Label	:= LblFunctions_SwitchingCommand;
//	Hysteresis	NEU NEU vorher Filter monitoring
	Hysteresis_PreAlarmLimitMAX         :FB_BA_Label	:= LblControl_PreAlarmLimitMAX;
    Hysteresis_PreAlarmLimitMIN         :FB_BA_Label	:= LblControl_PreAlarmLimitMIN;
    Hysteresis_PreAlarmFault            :FB_BA_Label	:= LblControl_PreAlarmFault;
    Hysteresis_MainAlarmLimitMAX        :FB_BA_Label	:= LblControl_MainAlarmLimitMAX;
    Hysteresis_MainAlarmLimitMIN        :FB_BA_Label	:= LblControl_MainAlarmLimitMIN;
    Hysteresis_MainAlarmFault           :FB_BA_Label	:= LblControl_MainAlarmFault;		
//	Monitoring	
	Monitoring_SwitchOnValue			:FB_BA_Label	:= LblFunctions_LimitMAX;
	Monitoring_SwitchOffValue			:FB_BA_Label	:= LblFunctions_LimitMIN;
	Monitoring_DelayFeedback			:FB_BA_Label	:= LblFunctions_FeedbackDelay;
	Monitoring_DelayInterruption		:FB_BA_Label	:= LblControl_TimeDelayInterruptionFeedback;
	Monitoring_Dst						:FB_BA_Label	:= LblFunctions_Fault;
	Monitoring_TiDly					:FB_BA_Label	:= LblControl_TimeDelay;
	Monitoring_HighLimitValue			:FB_BA_Label	:= LblFunctions_LimitMAX;
	Monitoring_LowLimitValue			:FB_BA_Label	:= LblFunctions_LimitMIN;
	Monitoring_HighLimitOn				:FB_BA_Label	:= LblFunctions_OperationalMessage;
	Monitoring_LowLimitOn				:FB_BA_Label	:= LblFunctions_OperationalMessage;
	Monitoring_Hys						:FB_BA_Label	:= LblFunctions_Hysteresis;
//	Operating Mode
	OperatingMode_OpModMan				:FB_BA_Label	:= LblControl_OperationModeSelection;	
	OperatingMode_OpModPr				:FB_BA_Label	:= LblControl_PresentOperationMode;		
	OperatingMode_Sched					:FB_BA_Label	:= LblFunctions_Scheduler;							
//	PID
	PID_Ctrl							:FB_BA_Label	:= LblFunctions_LoopObject;
	PID_Sp								:FB_BA_Label	:= LblFunctions_Setpoint;
//	FilterPT1	
	FilterPT1_DampingConstant			:FB_BA_Label	:= LblControl_DampConstant;
//	Ramp	
	Ramp_TiDown							:FB_BA_Label	:= LblControl_RampTimeDown;
	Ramp_TiUp							:FB_BA_Label	:= LblControl_RampTimeUp;
	Ramp_Y								:FB_BA_Label	:= LblFunctions_ControlSignal;
//	Scale
	Scale_X01							:FB_BA_Label	:= LblControl_X01;	
	Scale_X02							:FB_BA_Label	:= LblControl_X02;	
	Scale_X03							:FB_BA_Label	:= LblControl_X03;	
	Scale_X04							:FB_BA_Label	:= LblControl_X04;	
	Scale_X05							:FB_BA_Label	:= LblControl_X05;	
	Scale_X06							:FB_BA_Label	:= LblControl_X06;	
	Scale_X07							:FB_BA_Label	:= LblControl_X07;	
	
	Scale_Y01							:FB_BA_Label	:= LblControl_Y01;
	Scale_Y02							:FB_BA_Label	:= LblControl_Y02;
	Scale_Y03							:FB_BA_Label	:= LblControl_Y03;
	Scale_Y04							:FB_BA_Label	:= LblControl_Y04;
	Scale_Y05							:FB_BA_Label	:= LblControl_Y05;
	Scale_Y06							:FB_BA_Label	:= LblControl_Y06;
	Scale_Y07							:FB_BA_Label	:= LblControl_Y07;
	
	Scale_Ymin							:FB_BA_Label	:= LblFunctions_MinimumValue;
	Scale_Ymax							:FB_BA_Label	:= LblFunctions_MaximumValue;
	Scale_Y								:FB_BA_Label	:= LblFunctions_SetpointCalculated;
END_VAR

// ---- Templates/GVLs/DPAD/Labels/Composition/LblUniFieldDevice.TcGVL
{region '#Template'}
	{attribute 'Version' := '1.2.0.0'}
	{attribute 'Tags' := '"LCID": "1031", "Text": "GVL, Universal, AKS, Plants, ObjectName, Description"'}
	{attribute 'Tags' := '"LCID": "1033", "Text": "GVL, Universal, DPAD, Plants, ObjectName, Description"'}
	{attribute 'Description' := '"LCID": "1031", "Text": "Anlagenkennzeichnungssystem, Universal Labels Kompensation"'}
	{attribute 'Description' := '"LCID": "1033", "Text": "Data Point Addressing Description, Universal labels compensation"'}
{endregion}

{attribute 'qualified_only'}
// Universal Feldgeräte
VAR_GLOBAL
//	Universal\Aggregat
	Aggregat_Mdlt						:FB_BA_Label	:= LblFunctions_ControlSignal;
	Aggregat_Cmd						:FB_BA_Label	:= LblFunctions_SwitchingCommand;
	Aggregat_Dst						:FB_BA_Label	:= LblFunctions_Fault;
//	Universal\Damper	
	Dmp_SwiOpn							:FB_BA_Label	:= LblFunctions_FeedbackOPEN;
	Dmp_SwiCls							:FB_BA_Label	:= LblFunctions_FeedbackCLOSED;
	Dmp_Cmd								:FB_BA_Label	:= LblFunctions_SwitchingCommand;
	Dmp_Monit							:FB_BA_Label	:= LblControl_FeedbackMonitoring;
//	Universal\Motor	
	Motor_Dst							:FB_BA_Label	:= LblFunctions_Fault;
	Motor_Fdb							:FB_BA_Label	:= LblFunctions_Feedback;
	Motor_MntnSwi						:FB_BA_Label	:= LblFunctions_MaintenanceMessage;
	Motor_Monit							:FB_BA_Label	:= LblControl_FeedbackMonitoring;
	Motor_Cmd							:FB_BA_Label	:= LblFunctions_SwitchingCommand;
	Motor_Mdlt							:FB_BA_Label	:= LblFunctions_ControlSignal;
	Motor_Sp							:FB_BA_Label	:= LblFunctions_Setpoint;
	Motor_Ctrl							:FB_BA_Label	:= LblFunctions_LoopObject;
//	Universal\Pump
	Pump_DlyOff							:FB_BA_Label	:= LblControl_DelayOff;
	Pump_Ablk							:FB_BA_Label	:= LblControl_AntiBlocking;
	Pump_ThOvrld						:FB_BA_Label	:= LblFunctions_Fault;
	Pump_MntnSwi						:FB_BA_Label	:= LblFunctions_MaintenanceMessage;
	Pump_FlowSwi						:FB_BA_Label	:= LblControl_FlowSwitch;
	Pump_FlowMonit						:FB_BA_Label	:= LblAggregates_FlowMonitor;
//	Universal\Sensor
	SensorAnalog_MV_N					:FB_BA_Label	:= LblFunctions_MeasuredValueNorth;
	SensorAnalog_MV_S					:FB_BA_Label	:= LblFunctions_MeasuredValueSouth;
	SensorAnalog_MV_E					:FB_BA_Label	:= LblFunctions_MeasuredValueEast;
	SensorAnalog_MV_W					:FB_BA_Label	:= LblFunctions_MeasuredValueWest;
	SensorAnalog_MV						:FB_BA_Label	:= LblFunctions_MeasuredValue;
	SensorBinary_Input					:FB_BA_Label	:= LblFunctions_Fault;
	SensorButton_Input					:FB_BA_Label	:= LblFunctions_Button;
//	Universal\SmokeDetector	
	SmokeDetector_SmokeAlarm			:FB_BA_Label	:= LblControl_SmokeAlarm;
	SmokeDetector_SystemFailure			:FB_BA_Label	:= LblControl_SystemFailure;
	SmokeDetector_Contamination			:FB_BA_Label	:= LblControl_Contamination;
	SmokeDetector_AirFlow				:FB_BA_Label	:= LblControl_FlowSwitch;
	SmokeDetector_RstHw					:FB_BA_Label	:= LblControl_SwitchingCommandSmokeDetector;
	SmokeDetector_RstRm					:FB_BA_Label	:= LblControl_ButtonReset;
//	Universal\Valve	
	Valve_Ablk							:FB_BA_Label	:= LblControl_AntiBlocking;
	Valve_Fdb							:FB_BA_Label	:= LblFunctions_Feedback;
	Valve_Anlg3Pnt						:FB_BA_Label	:= LblControl_Converter3Point;
END_VAR

// ---- Templates/GVLs/EventClasses/EC_ID.TcGVL
{region '#Template'}
	{attribute 'Version' := '1.2.0.0'}
	{attribute 'Tags' := '"LCID": "1031", "Text": "General, Notification classes, Event classes, AMEV"'}
	{attribute 'Tags' := '"LCID": "1033", "Text": "General, Notification classes, Event classes, AMEV"'}
	{attribute 'Description' := '"LCID": "1031", "Text": "Ereignisklassen"'}
	{attribute 'Description' := '"LCID": "1033", "Text": "Event classes"'}
{endregion}

{attribute 'qualified_only'}
VAR_GLOBAL CONSTANT
	NC10							: UDINT := 10; // Gefahr für Leben // Danger to life	
	NC20							: UDINT := 20; // Sicherheitsmeldung // Safety message	
	NC30							: UDINT := 30; // Alarmeldung // Alarm message	
	NC40							: UDINT := 40; // Störungsmeldung // Fault message	
	NC50							: UDINT := 50; // Wartungsmeldung // Maintenance message	
	NC51							: UDINT := 51; // Wartungsmeldung // Maintenance message	
	NC60							: UDINT := 60; // Systemmeldung // System message	
	NC70							: UDINT := 70; // Handeingriff // Manual operation	
	NC80							: UDINT := 80; // Sonstige Meldungen // Other message	
END_VAR

// ---- Templates/GVLs/Language/English/LblAggregates_EN.TcGVL
{region '#Template'}
	{attribute 'Version' := '1.2.0.0'}
	{attribute 'Tags' := '"LCID": "1031", "Text": "GVL, AKS, Labels, ObjectName, Description"'}
	{attribute 'Tags' := '"LCID": "1033", "Text": "GVL, DPAD, Labels, ObjectName, Description"'}
	{attribute 'Description' := '"LCID": "1031", "Text": "Anlagenkennzeichnungssystem, Labels Aggregate"'}
	{attribute 'Description' := '"LCID": "1033", "Text": "Data Point Addressing Description, Labels aggregate"'}
{endregion}

{attribute 'global_init_slot' := '40510'}
VAR_GLOBAL
  LblAggregates_FunctionallyIndependentEequipment                 :FB_BA_Label:=( sObjName:='FIE',sDescr:='Functionally independent equipment');
  LblAggregates_SelfContainedControlUnit                          :FB_BA_Label:=( sObjName:='SCR',sDescr:='Self-contained control or regulation unit');
  LblAggregates_ControlCabinet                                    :FB_BA_Label:=( sObjName:='CCB',sDescr:='Control cabinet (trade-specific)');
//330 Doors, gates, windows, sun protection
  LblAggregates_WindowDrive                                       :FB_BA_Label:=( sObjName:='WIN',sDescr:='Window (drive)');
  LblAggregates_WindowContact                                     :FB_BA_Label:=( sObjName:='WIC',sDescr:='Window contact');
  LblAggregates_Blind                                             :FB_BA_Label:=( sObjName:='BLD',sDescr:='Blind');
  LblAggregates_Awning                                            :FB_BA_Label:=( sObjName:='AWN',sDescr:='Awning');
  LblAggregates_RollerShutters                                    :FB_BA_Label:=( sObjName:='ROS',sDescr:='Roller shutters');
  LblAggregates_Gate                                              :FB_BA_Label:=( sObjName:='GAT',sDescr:='Gate');
  LblAggregates_Door                                              :FB_BA_Label:=( sObjName:='DOR',sDescr:='Door');
  LblAggregates_DoorContact                                       :FB_BA_Label:=( sObjName:='DOC',sDescr:='Door contact');
  LblAggregates_Blackout                                          :FB_BA_Label:=( sObjName:='BLA',sDescr:='Blackout');
//412 Water plants
  LblAggregates_TraceHeating                                      :FB_BA_Label:=( sObjName:='THT',sDescr:='Trace heating');
  LblAggregates_ElectricHeating                                   :FB_BA_Label:=( sObjName:='EHT',sDescr:='Electric heating (warm water temperature preparation)');
  LblAggregates_WaterFilter                                       :FB_BA_Label:=( sObjName:='WFL',sDescr:='Water filter');
//421 Heat generation plants
  LblAggregates_Furnace                                           :FB_BA_Label:=( sObjName:='FUR',sDescr:='Furnace');
  LblAggregates_HeatExchanger                                     :FB_BA_Label:=( sObjName:='HEX',sDescr:='Heat exchanger');
//430 Ventilation and refrigeration systems
  LblAggregates_FanExhaustAir                                     :FB_BA_Label:=( sObjName:='EHF',sDescr:='Exhaust air fan');
  LblAggregates_Airwasher                                         :FB_BA_Label:=( sObjName:='AWA',sDescr:='Airwasher');
  LblAggregates_Humidifier                                        :FB_BA_Label:=( sObjName:='HUF',sDescr:='Humidifier');
  LblAggregates_HumidifierPump                                    :FB_BA_Label:=( sObjName:='HUP',sDescr:='Humidifier pump');
  LblAggregates_FireDamper                                        :FB_BA_Label:=( sObjName:='FID',sDescr:='Fire damper, fire protection valve');
  LblAggregates_SmokeProtectionDamper                             :FB_BA_Label:=( sObjName:='SPD',sDescr:='Smoke protection damper');
  LblAggregates_SmokeExtractorDamper                              :FB_BA_Label:=( sObjName:='SEP',sDescr:='Smoke extractor damper');
  LblAggregates_CeilingSwirlDiffuser                              :FB_BA_Label:=( sObjName:='CSD',sDescr:='Ceiling swirl diffuser');
  LblAggregates_RoofAirHeater                                     :FB_BA_Label:=( sObjName:='RAH',sDescr:='Roof air heater');
  LblAggregates_DirectEvaporator                                  :FB_BA_Label:=( sObjName:='DEA',sDescr:='Direct evaporator');
  LblAggregates_ElectricalAirHeater                               :FB_BA_Label:=( sObjName:='EAH',sDescr:='Electrical air heater');
  LblAggregates_ElectricReHeater                                  :FB_BA_Label:=( sObjName:='ERH',sDescr:='Electric re-heater');
  LblAggregates_ElectricaPreHeater                                :FB_BA_Label:=( sObjName:='EPH',sDescr:='Electrical pre-heater');
  LblAggregates_HeaterGeneral                                     :FB_BA_Label:=( sObjName:='HTR',sDescr:='Heater ');
  LblAggregates_FanExtractAir                                     :FB_BA_Label:=( sObjName:='EXF',sDescr:='Extract air fan ');
  LblAggregates_InductionDevice                                   :FB_BA_Label:=( sObjName:='IND',sDescr:='Induction device');
  LblAggregates_RefrigerantDryer                                  :FB_BA_Label:=( sObjName:='RFD',sDescr:='Refrigerant dryer');
  LblAggregates_CirculatorySystem                                 :FB_BA_Label:=( sObjName:='CCS',sDescr:='Circulatory system ');
  LblAggregates_AirFilterOutsideAir                               :FB_BA_Label:=( sObjName:='AFI',sDescr:='Outside air filter');
  LblAggregates_AirFilterSupplyAir                                :FB_BA_Label:=( sObjName:='AFI',sDescr:='Supply air filter');
  LblAggregates_AirFilterExhaustAir                               :FB_BA_Label:=( sObjName:='AFI',sDescr:='Exhaus air filter');
  LblAggregates_AirFilterExtractAir                               :FB_BA_Label:=( sObjName:='AFI',sDescr:='Extract air filter');
  LblAggregates_AirFilter                                         :FB_BA_Label:=( sObjName:='AFI',sDescr:='Air filter');
  LblAggregates_VentilationDamper                                 :FB_BA_Label:=( sObjName:='VFL',sDescr:='Ventilation flap');
  LblAggregates_VentilationDamperOutsideAir                       :FB_BA_Label:=( sObjName:='VFL',sDescr:='Ventilation flap outside air');
  LblAggregates_VentilationDamperExhaustAir                       :FB_BA_Label:=( sObjName:='VFL',sDescr:='Ventilation flap exhaust air');
  LblAggregates_VentilationDamperMixAir                           :FB_BA_Label:=( sObjName:='VFL',sDescr:='Ventilation flap mix air');
  LblAggregates_VentilationDamperSupplyAir                        :FB_BA_Label:=( sObjName:='VFL',sDescr:='Ventilation flap supply air');
  LblAggregates_VentilationDamperBypassAir                        :FB_BA_Label:=( sObjName:='VFL',sDescr:='Ventilation flap bypass');
  LblAggregates_Pump                                              :FB_BA_Label:=( sObjName:='PUM',sDescr:='Pump');
  LblAggregates_RecirculatingAirCoolingDevice                     :FB_BA_Label:=( sObjName:='RAC',sDescr:='Recirculating air cooling device');
  LblAggregates_FanRecirculatingAir                               :FB_BA_Label:=( sObjName:='RAF',sDescr:='Recirculating air fan');
  LblAggregates_UvFilter                                          :FB_BA_Label:=( sObjName:='UVF',sDescr:='UV filter');
  LblAggregates_VariableFlowRateController                        :FB_BA_Label:=( sObjName:='VFC',sDescr:='Variable flow rate controller');
  LblAggregates_WaterAirHeater                                    :FB_BA_Label:=( sObjName:='WAH',sDescr:='Water air heater');
  LblAggregates_WaterReHeater                                     :FB_BA_Label:=( sObjName:='WRH',sDescr:='Water re-heater');
  LblAggregates_WaterPreHeater                                    :FB_BA_Label:=( sObjName:='WPH',sDescr:='Water pre-heater');
  LblAggregates_HeatRecovery                                      :FB_BA_Label:=( sObjName:='HRC',sDescr:='Heat recovery');
  LblAggregates_FanSupplyAir                                      :FB_BA_Label:=( sObjName:='SUF',sDescr:='Supply air fan');
  LblAggregates_SmokeExtractionSystems                            :FB_BA_Label:=( sObjName:='SES',sDescr:='Smoke extraction systems');
  LblAggregates_SmokeExtractionVentilator                         :FB_BA_Label:=( sObjName:='SEF',sDescr:='Smoke extraction fan');
  LblAggregates_VentWindow                                        :FB_BA_Label:=( sObjName:='VWI',sDescr:='Vent window');
  LblAggregates_VentFlap                                          :FB_BA_Label:=( sObjName:='VFL',sDescr:='Vent flap');
  LblAggregates_VentDoor                                          :FB_BA_Label:=( sObjName:='VDO',sDescr:='Vent door');
  LblAggregates_WakeFan                                           :FB_BA_Label:=( sObjName:='WAF',sDescr:='Wake fan');
//434 Refrigeration systems
  LblAggregates_GlycoOilProtector                                 :FB_BA_Label:=( sObjName:='GLP',sDescr:='Glycol/oil protector');
  LblAggregates_Chiller                                           :FB_BA_Label:=( sObjName:='CHI',sDescr:='Chiller');
  LblAggregates_ReCoolingPlant                                    :FB_BA_Label:=( sObjName:='RCP',sDescr:='Re-cooling plant');
//440 High-voltage systems
  LblAggregates_GeneralPowerSupply                                :FB_BA_Label:=( sObjName:='GPS',sDescr:='General power supply');
  LblAggregates_CombindeHeatPowerStation                          :FB_BA_Label:=( sObjName:='CGU',sDescr:='Co-generation unit');
  LblAggregates_CompensationSystem                                :FB_BA_Label:=( sObjName:='CPS',sDescr:='Compensation system');
  LblAggregates_CouplingSwitch                                    :FB_BA_Label:=( sObjName:='COS',sDescr:='Coupling switch');
  LblAggregates_LoadBreakSwitch                                   :FB_BA_Label:=( sObjName:='LBS',sDescr:='Load-break switch');
  LblAggregates_CircuitBreaker                                    :FB_BA_Label:=( sObjName:='CCB',sDescr:='Circuit breaker');
  LblAggregates_NetworkAnalyser                                   :FB_BA_Label:=( sObjName:='NWA',sDescr:='Network analyser');
  LblAggregates_EmergencyPoweGeneratorUnit                        :FB_BA_Label:=( sObjName:='EPG',sDescr:='Emergency power generator unit');
  LblAggregates_EmergencyLighting                                 :FB_BA_Label:=( sObjName:='EML',sDescr:='Emergency lighting');
  LblAggregates_SafetyPowerSupply                                 :FB_BA_Label:=( sObjName:='SPS',sDescr:='Safety power supply');
  LblAggregates_Transformer                                       :FB_BA_Label:=( sObjName:='TRF',sDescr:='Transformer');
  LblAggregates_UninterruptiblePowerSupply                        :FB_BA_Label:=( sObjName:='UPS',sDescr:='Uninterruptible power supply');
//450 Telecommunications and information technology equipment
  LblAggregates_CentralFireAlarmSystem                            :FB_BA_Label:=( sObjName:='CFA',sDescr:='Central fire alarm system');
  LblAggregates_FireControlPanel                                  :FB_BA_Label:=( sObjName:='FCP',sDescr:='Fire control panel');
  LblAggregates_KitchenTableau                                    :FB_BA_Label:=( sObjName:='KIT',sDescr:='Kitchen tableau');
  LblAggregates_SmokeDetector                                     :FB_BA_Label:=( sObjName:='SDE',sDescr:='Smoke detector');
  LblAggregates_SmokeProtectionScreen                             :FB_BA_Label:=( sObjName:='SPS',sDescr:='Smoke protection screen');
  LblAggregates_VoiceAlarmCentre                                  :FB_BA_Label:=( sObjName:='VAC',sDescr:='Voice alarm centre');
  LblAggregates_Tableau                                           :FB_BA_Label:=( sObjName:='TAB',sDescr:='Tableau (general)');
//460 Conveyors
  LblAggregates_LiftGeneral                                       :FB_BA_Label:=( sObjName:='LIG',sDescr:='Lift general');
  LblAggregates_GoodsLift                                         :FB_BA_Label:=( sObjName:='GLI',sDescr:='Goods lift');
  LblAggregates_PassengerLift                                     :FB_BA_Label:=( sObjName:='PLI',sDescr:='Passenger lift');
//470 User-specific systems
  LblAggregates_FumeCupboard                                      :FB_BA_Label:=( sObjName:='FCB',sDescr:='Fume cupboard');
  LblAggregates_Compressor                                        :FB_BA_Label:=( sObjName:='COM',sDescr:='Compressor');
  LblAggregates_ProgrammableLogicControllers                      :FB_BA_Label:=( sObjName:='PLC',sDescr:='Programmable logic controllers');
//479 User-specific system, weather station
  LblAggregates_RainSensor                                        :FB_BA_Label:=( sObjName:='RAS',sDescr:='Rain sensor');
  LblAggregates_SolarRadiation                                    :FB_BA_Label:=( sObjName:='SOR',sDescr:='Solar radiation');
  LblAggregates_WeatherStation                                    :FB_BA_Label:=( sObjName:='WST',sDescr:='Weather station');
  LblAggregates_WindSpeed                                         :FB_BA_Label:=( sObjName:='WIS',sDescr:='Wind speed');
  LblAggregates_WindDirection                                     :FB_BA_Label:=( sObjName:='WID',sDescr:='Wind direction');
  LblAggregates_WindForce                                         :FB_BA_Label:=( sObjName:='WDF',sDescr:='Wind force');
  LblAggregates_Brightness                                        :FB_BA_Label:=( sObjName:='BIN',sDescr:='Brightness');
  LblAggregates_Dawn                                              :FB_BA_Label:=( sObjName:='BID',sDescr:='Brightness dawn');
  LblAggregates_PressureAbsolute                                  :FB_BA_Label:=( sObjName:='PAB',sDescr:='Pressure absolute');
  LblAggregates_PressureRelative                                  :FB_BA_Label:=( sObjName:='PRE',sDescr:='Pressure relative');
  LblAggregates_GeoLatitude                                       :FB_BA_Label:=( sObjName:='LAT',sDescr:='Latitude       ');
  LblAggregates_GeoLongitude                                      :FB_BA_Label:=( sObjName:='LOT',sDescr:='Longitude      ');
  LblAggregates_SunAzimuth                                        :FB_BA_Label:=( sObjName:='AZI',sDescr:='Azimuth        ');
  LblAggregates_SunElevation                                      :FB_BA_Label:=( sObjName:='ELE',sDescr:='Elevation      ');
//480 Building automation and control systems
  LblAggregates_SystemSwitch                                      :FB_BA_Label:=( sObjName:='SYS',sDescr:='System switch');
  LblAggregates_AutomationStationEquipment                        :FB_BA_Label:=( sObjName:='ASE',sDescr:='Automation station equipment');
  LblAggregates_BusLineCoupler                                    :FB_BA_Label:=( sObjName:='BUS',sDescr:='Bus line coupler');
  LblAggregates_DataInterfaceUnit                                 :FB_BA_Label:=( sObjName:='DIU',sDescr:='Data interface unit');
  LblAggregates_FieldbusModule                                    :FB_BA_Label:=( sObjName:='FBM',sDescr:='Fieldbus module');
  LblAggregates_InformationFocalPoint                             :FB_BA_Label:=( sObjName:='IFP',sDescr:='Information focal point');
  LblAggregates_ManagementAndControlEquipment                     :FB_BA_Label:=( sObjName:='MCE',sDescr:='Management and control equipment');
//481 BACS sensors – temperature
  LblAggregates_TemperatureGasEmission                            :FB_BA_Label:=( sObjName:='TEG',sDescr:='Emissions gas temperature');
  LblAggregates_TemperatureExtractAir                             :FB_BA_Label:=( sObjName:='TEX',sDescr:='Extract air temperature');
  LblAggregates_TemperatureOutside                                :FB_BA_Label:=( sObjName:='TOU',sDescr:='Outside temperature');
  LblAggregates_TemperatureExhaustAir                             :FB_BA_Label:=( sObjName:='TEH',sDescr:='Exhaust air temperature');
  LblAggregates_FrostProtectionMonitor                            :FB_BA_Label:=( sObjName:='FPM',sDescr:='Frost protection monitor');
  LblAggregates_TemperatureMixedAir                               :FB_BA_Label:=( sObjName:='TMI',sDescr:='Mixed air temperature');
  LblAggregates_TemperatureRoomAir                                :FB_BA_Label:=( sObjName:='TRO',sDescr:='Room temperature');
  LblAggregates_TemperatureReturnFlow                             :FB_BA_Label:=( sObjName:='TRT',sDescr:='Return flow temperature');
  LblAggregates_LimiterSafetyTemperature                          :FB_BA_Label:=( sObjName:='STL',sDescr:='Safety temperature limiter');
  LblAggregates_MonitorSafetyTemperature                          :FB_BA_Label:=( sObjName:='STM',sDescr:='Safety temperature monitor');
  LblAggregates_TemperatureStorage                                :FB_BA_Label:=( sObjName:='TST',sDescr:='Storage temperature');
  LblAggregates_TemperatureDewPoint                               :FB_BA_Label:=( sObjName:='TDP',sDescr:='Dew point temperature');
  LblAggregates_MonitorDewPoint                                   :FB_BA_Label:=( sObjName:='DPM',sDescr:='Dew point monitor');
  LblAggregates_TemperatureAfterCooler                            :FB_BA_Label:=( sObjName:='TAC',sDescr:='Temperature after cooler');
  LblAggregates_TemperatureAfterPreHeater                         :FB_BA_Label:=( sObjName:='TAP',sDescr:='Temperature after pre-heater');
  LblAggregates_TemperatureAfterHeatRecovery                      :FB_BA_Label:=( sObjName:='TAR',sDescr:='Temperature after heat recovery');
  LblAggregates_Thermostat                                        :FB_BA_Label:=( sObjName:='THM',sDescr:='Thermostat');
  LblAggregates_TemperatureHotWater                               :FB_BA_Label:=( sObjName:='THW',sDescr:='Hot water temperature');
  LblAggregates_TemperatureCirculation                            :FB_BA_Label:=( sObjName:='TCI',sDescr:='Circulation temperature');
  LblAggregates_TemperatureRecirculatingAir                       :FB_BA_Label:=( sObjName:='TRE',sDescr:='Recirculating air temperature');
  LblAggregates_TemperatureFlow                                   :FB_BA_Label:=( sObjName:='TFL',sDescr:='Flow temperature');
  LblAggregates_TemperatureSupplyAir                              :FB_BA_Label:=( sObjName:='TSU',sDescr:='Supply air temperature');
//481 BACS sensors – pressure
  LblAggregates_PressureExtractAir                                :FB_BA_Label:=( sObjName:='PEX',sDescr:='Extract air pressure');
  LblAggregates_PressureOutsideAir                                :FB_BA_Label:=( sObjName:='POU',sDescr:='Outside air pressure');
  LblAggregates_PressureDifferential                              :FB_BA_Label:=( sObjName:='PDI',sDescr:='Differential pressure');
  LblAggregates_PressureDifferentialOutsideAirFilter              :FB_BA_Label:=( sObjName:='PDI',sDescr:='Differential pressure outside air filter');
  LblAggregates_PressureDifferentialExtractAirFilter              :FB_BA_Label:=( sObjName:='PDI',sDescr:='Differential pressure extract air filter');
  LblAggregates_PressureDifferentialExhaustAirFilter              :FB_BA_Label:=( sObjName:='PDI',sDescr:='Differential pressure exhaust air filter');
  LblAggregates_PressureDifferentialSupplyAirFan                  :FB_BA_Label:=( sObjName:='PDI',sDescr:='Differential pressure supply air fan');
  LblAggregates_PressureDifferentialExtractAirFan                 :FB_BA_Label:=( sObjName:='PDI',sDescr:='Differential pressure ectract air fan');
  LblAggregates_PressureDifferentialExhaustAirFan                 :FB_BA_Label:=( sObjName:='PDI',sDescr:='Differential pressure exhaust air fan');
  LblAggregates_PressureSensorFlow                                :FB_BA_Label:=( sObjName:='PFL',sDescr:='Pressure sensor (water) flow');
  LblAggregates_MonitorPressure                                   :FB_BA_Label:=( sObjName:='PCO',sDescr:='Pressure controller');
  LblAggregates_PressureExhaustAir                                :FB_BA_Label:=( sObjName:='PEH',sDescr:='Exhaust air pressure');
  LblAggregates_PressureRoomAir                                   :FB_BA_Label:=( sObjName:='PRO',sDescr:='Room pressure');
  LblAggregates_PressureIndexCircuitSensorDifferential            :FB_BA_Label:=( sObjName:='PSI',sDescr:='Index circuit sensor differential pressure');
  LblAggregates_LimiterSafetyPressure                             :FB_BA_Label:=( sObjName:='SPL',sDescr:='Safety pressure limiter');
  LblAggregates_PressureSupplyAir                                 :FB_BA_Label:=( sObjName:='PSU',sDescr:='Supply air pressure');
//481 BACS sensors – air quality
  LblAggregates_CO2Sensor                                         :FB_BA_Label:=( sObjName:='COM',sDescr:='CO2 sensor');
  LblAggregates_QualityExtractAir                                 :FB_BA_Label:=( sObjName:='QEX',sDescr:='Extract air quality');
  LblAggregates_OualityRoomAir                                    :FB_BA_Label:=( sObjName:='QRO',sDescr:='Room air quality');
  LblAggregates_QualitiySupplyAir                                 :FB_BA_Label:=( sObjName:='QSU',sDescr:='Supply air quality');
  LblAggregates_QualityAirSensor                                  :FB_BA_Label:=( sObjName:='AQS',sDescr:='Air quality sensor');
//481 BACS sensors – humidity
  LblAggregates_Hygrostat                                         :FB_BA_Label:=( sObjName:='HYG',sDescr:='Hygrostat');
  LblAggregates_RelativeHumiditiyExtractAir                       :FB_BA_Label:=( sObjName:='HEX',sDescr:='Relative extract air humidity');
  LblAggregates_RelativeHumidityOutsideAir                        :FB_BA_Label:=( sObjName:='HOU',sDescr:='Relative outside air humidity');
  LblAggregates_RelativeHumidityExhaustAir                        :FB_BA_Label:=( sObjName:='HEH',sDescr:='Relative exhaust air humidity');
  LblAggregates_MonitorCondensation                               :FB_BA_Label:=( sObjName:='HCM',sDescr:='Condensation monitor');
  LblAggregates_RelativeHumidityMixedAir                          :FB_BA_Label:=( sObjName:='HMI',sDescr:='Relative mixed air humidity');
  LblAggregates_RelativeHumidityRoomHumidity                      :FB_BA_Label:=( sObjName:='HRO',sDescr:='Relative room humidity');
  LblAggregates_RelativeHumidityRecirculatedAir                   :FB_BA_Label:=( sObjName:='HRE',sDescr:='Relative recirculated air humidity');
  LblAggregates_RelativeHumiditySupplyAir                         :FB_BA_Label:=( sObjName:='HSU',sDescr:='Relative supply air humidity');
  LblAggregates_AbsoluteHumidityExtractAir                        :FB_BA_Label:=( sObjName:='XEX',sDescr:='Absolute extract air humidity');
  LblAggregates_AbsoluteHumidtiyOutsideAir                        :FB_BA_Label:=( sObjName:='XOU',sDescr:='Absolute outsie air humidity');
  LblAggregates_AbsoluteHumidtiyExhaustAir                        :FB_BA_Label:=( sObjName:='XEH',sDescr:='Absolute exhaust air humidity');
  LblAggregates_AbsoluteHumidityMixedAir                          :FB_BA_Label:=( sObjName:='XMI',sDescr:='Absolute mixed air humidity');
  LblAggregates_AbsoluteHumidityRoomAir                           :FB_BA_Label:=( sObjName:='XRO',sDescr:='Absolute room humidity');
  LblAggregates_AbsoluteHumidityRecirculatingAir                  :FB_BA_Label:=( sObjName:='XRE',sDescr:='Absolute recirculating air humidity');
  LblAggregates_AbsoluteHumiditySupplyAir                         :FB_BA_Label:=( sObjName:='XSU',sDescr:='Absolute supply air humidity');
//481 BACS sensors – consumption recording
  LblAggregates_MeterElectric                                     :FB_BA_Label:=( sObjName:='ELM',sDescr:='Electric meter');
  LblAggregates_MeterGasNaturalGas                                :FB_BA_Label:=( sObjName:='GAM',sDescr:='Gas meter natural gas');
  LblAggregates_MeterCoolingEnergy                                :FB_BA_Label:=( sObjName:='CEM',sDescr:='Cooling energy meter');
  LblAggregates_MeterHeat                                         :FB_BA_Label:=( sObjName:='HEM',sDescr:='Heat meter');
  LblAggregates_MetferWater                                       :FB_BA_Label:=( sObjName:='WAM',sDescr:='Water meter');
  LblAggregates_MeterFuel                                         :FB_BA_Label:=( sObjName:='FUM',sDescr:='Fuel meter (oil)');
  LblAggregates_MeterSteam                                        :FB_BA_Label:=( sObjName:='STM',sDescr:='Steam meter');
  LblAggregates_DegreeDayNumber                                   :FB_BA_Label:=( sObjName:='DDN',sDescr:='Degree day number');
//481 BACS sensors – condition recording and other
  LblAggregates_LeakageMonitoring                                 :FB_BA_Label:=( sObjName:='LKM',sDescr:='Leakage monitoring');
  LblAggregates_EmergencyStop                                     :FB_BA_Label:=( sObjName:='EMG',sDescr:='Emergency stop unit/button');
  LblAggregates_StockLevel                                        :FB_BA_Label:=( sObjName:='SLV',sDescr:='Stock level');
  LblAggregates_FlowMonitor                                       :FB_BA_Label:=( sObjName:='FLM',sDescr:='Flow monitor');
  LblAggregates_OverflowMonitoring                                :FB_BA_Label:=( sObjName:='OVM',sDescr:='Overflow monitoring');
  LblAggregates_LowWaterCutOff                                    :FB_BA_Label:=( sObjName:='WCO',sDescr:='Low-water cut-off');
  LblAggregates_WaterFlowMonitor                                  :FB_BA_Label:=( sObjName:='WFM',sDescr:='Water flow monitor');
//481 BACS sensors – speed
  LblAggregates_PumpSpeed                                         :FB_BA_Label:=( sObjName:='SPU',sDescr:='Pump speed');
  LblAggregates_FanSpeedExtractAir                                :FB_BA_Label:=( sObjName:='SEX',sDescr:='Fan speed (extract air)');
  LblAggregates_FanSpeedExhaustAir                                :FB_BA_Label:=( sObjName:='SEH',sDescr:='Fan speed (exhaust air)');
  LblAggregates_FanSpeedSupplyAir                                 :FB_BA_Label:=( sObjName:='SSU',sDescr:='Fan speed (supply air)');
//481 BACS sensors – volume flow
  LblAggregates_VolumeFlowRateExtractAir                          :FB_BA_Label:=( sObjName:='VEX',sDescr:='Extract air volume flow rate');
  LblAggregates_VolumeFlowRateOutsideAir                          :FB_BA_Label:=( sObjName:='VOU',sDescr:='Outside air volume flow rate');
  LblAggregates_VolumeFlowRateExhaustAir                          :FB_BA_Label:=( sObjName:='VEH',sDescr:='Exhaust air volume flow rate');
  LblAggregates_VolumeFlowRateBrineCirculatorySystem              :FB_BA_Label:=( sObjName:='VBR',sDescr:='Volume flow brine (circulatory system)');
  LblAggregates_VolumeFlowRateColdDrinkingWater                   :FB_BA_Label:=( sObjName:='VCW',sDescr:='Volume flow cold drinking water');
  LblAggregates_VolumeFlowRateHotDrinkingWater                    :FB_BA_Label:=( sObjName:='VHW',sDescr:='Volume flow hot drinking water');
  LblAggregates_VolumeFlowRateWaterPurification                   :FB_BA_Label:=( sObjName:='VWP',sDescr:='Volume flow water purification');
  LblAggregates_VolumeFlowRateSupplyAir                           :FB_BA_Label:=( sObjName:='VSU',sDescr:='Supply air volume flow');
//481 BACS actuators – actuating drives
  LblAggregates_ValveRadiator                                     :FB_BA_Label:=( sObjName:='RDV',sDescr:='Radiator valve drive');
  LblAggregates_ValveCoolingCeiling                               :FB_BA_Label:=( sObjName:='CCV',sDescr:='Cooling ceiling valve drive');
  LblAggregates_MotorisedFlap                                     :FB_BA_Label:=( sObjName:='FLA',sDescr:='Motorised flap');
  LblAggregates_Valve                                             :FB_BA_Label:=( sObjName:='VLV',sDescr:='Motor valve');
  LblAggregates_HumidifierValve                                   :FB_BA_Label:=( sObjName:='VLV',sDescr:='Humidifier valve');
//481 BACS lighting
  LblAggregates_IlluminationExternal                              :FB_BA_Label:=( sObjName:='EOU',sDescr:='Illumination outside');
  LblAggregates_IlluminationRoom                                  :FB_BA_Label:=( sObjName:='ERO',sDescr:='Illumination room');
  LblAggregates_LightColourRoom                                   :FB_BA_Label:=( sObjName:='CRO',sDescr:='Light colour room');
  LblAggregates_RedLightIntensity                                 :FB_BA_Label:=( sObjName:='LRD',sDescr:='Red light intensity');
  LblAggregates_GreenLightIntensity                               :FB_BA_Label:=( sObjName:='LGN',sDescr:='Green light intensity');
  LblAggregates_BlueLightIntensity                                :FB_BA_Label:=( sObjName:='LBL',sDescr:='Blue light intensity');
//481 BACS sun protection
  LblAggregates_BlindAnglePosition                                :FB_BA_Label:=( sObjName:='BAP',sDescr:='Blind angle position');
  LblAggregates_ShadingPosition                                   :FB_BA_Label:=( sObjName:='BSP',sDescr:='Shading position');
  LblAggregates_MovementCommand                                   :FB_BA_Label:=( sObjName:='BMC',sDescr:='Blind Movement command');
//485 Room automation
  LblAggregates_DisplayAndControlUnit                             :FB_BA_Label:=( sObjName:='DCU',sDescr:='Display and control unit');
  LblAggregates_PresenceSwitches                                  :FB_BA_Label:=( sObjName:='PDE',sDescr:='Presence switches, detectors, motion detectors');
  LblAggregates_RoomAutomationDevice                              :FB_BA_Label:=( sObjName:='RAD',sDescr:='Room automation device');
  LblAggregates_RoomControlUnit                                   :FB_BA_Label:=( sObjName:='RCU',sDescr:='Room control unit');
END_VAR

// ---- Templates/GVLs/Language/English/LblControl_EN.TcGVL
{region '#Template'}
	{attribute 'Version' := '1.2.0.0'}
	{attribute 'Tags' := '"LCID": "1031", "Text": "GVL, AKS, Labels, ObjectName, Description"'}
	{attribute 'Tags' := '"LCID": "1033", "Text": "GVL, DPAD, Labels, ObjectName, Description"'}
	{attribute 'Description' := '"LCID": "1031", "Text": "Anlagenkennzeichnungssystem, Labels controls"'}
	{attribute 'Description' := '"LCID": "1033", "Text": "Data Point Addressing Description, Labels controls"'}
{endregion}
	 
